Staubli VAL3: OnF1.pgx

program OnF1()
begin
  //
  switch nPage
    //初始化砂带
    case 0
      call InitBelt()
      bUserRefresh=true
    break
    //暂停
    case 1
      if !bPause
        stopMove()
        bPause=true
        call Message("运动暂停",true)
      else
        restartMove()
        bPause=false
        call Message("运动继续",true)
      endIf
    break

  endSwitch
end
